FUNCTION_BLOCK E_TP (* standard timer function block (pulse) *)
  (* Standard: 61499-2; Classification: standard timer function block *)
  (* Version 1.0, 2024-03-04, franz *)
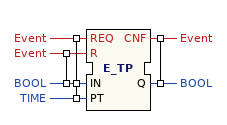
  EVENT_INPUT
    REQ WITH IN, PT; (* Service Request *)
    R WITH IN; (* Reset *)
  END_EVENT
  EVENT_OUTPUT
    CNF WITH Q; (* Confirmation of Requested Service *)
  END_EVENT
  VAR_INPUT
    IN : BOOL; (* Input *)
    PT : TIME; (* Pulse time *)
  END_VAR
  VAR_OUTPUT
    Q : BOOL; (* Output *)
  END_VAR
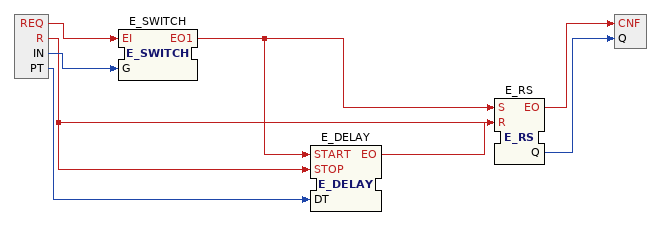
  FBS
    E_SWITCH : E_SWITCH;
    E_DELAY : E_DELAY;
    E_RS : E_RS;
  END_FBS
  EVENT_CONNECTIONS
    REQ TO E_SWITCH.EI;
    E_RS.EO TO CNF;
    E_SWITCH.EO1 TO E_DELAY.START;
    E_SWITCH.EO1 TO E_RS.S;
    R TO E_DELAY.STOP;
    R TO E_RS.R;
    E_DELAY.EO TO E_RS.R;
  END_CONNECTIONS
  DATA_CONNECTIONS
    IN TO E_SWITCH.G;
    PT TO E_DELAY.DT;
    E_RS.Q TO Q;
  END_CONNECTIONS
END_FUNCTION_BLOCK
